Universal Robots URScript: script_ur5e.urscript

def ur5e_dibujar():
  textmsg("=== UR5e: inicio del programa ===")
  q_home = get_actual_joint_positions()
  textmsg("UR5e HOME guardado")
  # === Ir al origen calibrado: UR5e ===
  textmsg("UR5e - yendo al origen calibrado")
  x0 = 0.68387
  y0 = -0.03000
  z_mesa = 0.00221
  rx = 2.48100
  ry = -1.92700
  rz = 0.00000
  # Primero se acerca por arriba; nunca va directamente a la Z baja.
  movel(p[x0, y0, z_mesa+0.06000, rx, ry, rz], a=0.03, v=0.05)
  sleep(0.3)
  # === Detección única de superficie por fuerza: UR5e ===
  textmsg("UR5e - Detectando superficie una sola vez...")
  zero_ftsensor()
  sleep(0.5)
  i_f = 0
  while (force() < 2.000 and i_f < 2000):
    speedl([0, 0, -0.00800, 0, 0, 0], 0.25, 0.02)
    i_f = i_f + 1
  end
  stopl(3.0)
  sleep(0.2)
  if (i_f >= 2000):
    popup("UR5e: No se detectó superficie. Revisa posición inicial y F_UMBRAL.", error=True)
    halt
  end
  z_contacto = get_actual_tcp_pose()[2]
  z_dibujo = z_contacto + 0.00150
  textmsg("UR5e - z_contacto=", z_contacto)
  textmsg("UR5e - z_dibujo=", z_dibujo)
  movel(p[x0, y0, z_dibujo+0.02500, rx, ry, rz], a=0.03, v=0.04)
  sleep(0.2)
  # === Dibujo - UR5e - 3 trazos ===

  # --- Trazo 1 / 3 ---
  textmsg("UR5e - Trazo 1 de 3")
  movel(p[x0+0.01300, y0+-0.00696, z_dibujo+0.02500, rx, ry, rz], a=0.03, v=0.04)
  movel(p[x0+0.01300, y0+-0.00696, z_dibujo, rx, ry, rz], a=0.006, v=0.002)
  movel(p[x0+0.01269, y0+-0.00665, z_dibujo, rx, ry, rz], a=0.008, v=0.025, r=0.0002)
  movel(p[x0+0.01114, y0+-0.00665, z_dibujo, rx, ry, rz], a=0.008, v=0.025, r=0.0002)
  movel(p[x0+0.00990, y0+-0.00882, z_dibujo, rx, ry, rz], a=0.008, v=0.025, r=0.0002)
  movel(p[x0+0.00743, y0+-0.01130, z_dibujo, rx, ry, rz], a=0.008, v=0.025, r=0.0002)
  movel(p[x0+0.00464, y0+-0.01285, z_dibujo, rx, ry, rz], a=0.008, v=0.025, r=0.0002)
  movel(p[x0+0.00155, y0+-0.01346, z_dibujo, rx, ry, rz], a=0.008, v=0.025, r=0.0002)
  movel(p[x0+0.00124, y0+-0.01377, z_dibujo, rx, ry, rz], a=0.008, v=0.025, r=0.0002)
  movel(p[x0+0.00124, y0+-0.02182, z_dibujo, rx, ry, rz], a=0.008, v=0.025, r=0.0002)
  movel(p[x0+0.00217, y0+-0.02430, z_dibujo, rx, ry, rz], a=0.008, v=0.025, r=0.0002)
  movel(p[x0+0.00557, y0+-0.02801, z_dibujo, rx, ry, rz], a=0.008, v=0.025, r=0.0002)
  movel(p[x0+0.00960, y0+-0.02956, z_dibujo, rx, ry, rz], a=0.008, v=0.025, r=0.0002)
  movel(p[x0+0.01238, y0+-0.02956, z_dibujo, rx, ry, rz], a=0.008, v=0.025, r=0.0002)
  movel(p[x0+0.01269, y0+-0.02925, z_dibujo, rx, ry, rz], a=0.008, v=0.025, r=0.0002)
  movel(p[x0+0.01486, y0+-0.02894, z_dibujo, rx, ry, rz], a=0.008, v=0.025, r=0.0002)
  movel(p[x0+0.01888, y0+-0.02677, z_dibujo, rx, ry, rz], a=0.008, v=0.025, r=0.0002)
  movel(p[x0+0.02229, y0+-0.02306, z_dibujo, rx, ry, rz], a=0.008, v=0.025, r=0.0002)
  movel(p[x0+0.02383, y0+-0.01935, z_dibujo, rx, ry, rz], a=0.008, v=0.025, r=0.0002)
  movel(p[x0+0.02383, y0+-0.01532, z_dibujo, rx, ry, rz], a=0.008, v=0.025, r=0.0002)
  movel(p[x0+0.02229, y0+-0.01192, z_dibujo, rx, ry, rz], a=0.008, v=0.025, r=0.0002)
  movel(p[x0+0.01888, y0+-0.00882, z_dibujo, rx, ry, rz], a=0.008, v=0.025, r=0.0002)
  movel(p[x0+0.01331, y0+-0.00696, z_dibujo, rx, ry, rz], a=0.008, v=0.025, r=0.0002)
  movel(p[x0+0.01331, y0+-0.00696, z_dibujo+0.02500, rx, ry, rz], a=0.03, v=0.04)

  # --- Trazo 2 / 3 ---
  textmsg("UR5e - Trazo 2 de 3")
  movel(p[x0+0.02198, y0+0.01625, z_dibujo+0.02500, rx, ry, rz], a=0.03, v=0.04)
  movel(p[x0+0.02198, y0+0.01625, z_dibujo, rx, ry, rz], a=0.006, v=0.002)
  movel(p[x0+0.02167, y0+0.01656, z_dibujo, rx, ry, rz], a=0.008, v=0.025, r=0.0002)
  movel(p[x0+0.01733, y0+0.01656, z_dibujo, rx, ry, rz], a=0.008, v=0.025, r=0.0002)
  movel(p[x0+0.01455, y0+0.01532, z_dibujo, rx, ry, rz], a=0.008, v=0.025, r=0.0002)
  movel(p[x0+0.01269, y0+0.01377, z_dibujo, rx, ry, rz], a=0.008, v=0.025, r=0.0002)
  movel(p[x0+0.00836, y0+0.00789, z_dibujo, rx, ry, rz], a=0.008, v=0.025, r=0.0002)
  movel(p[x0+0.00836, y0+0.00727, z_dibujo, rx, ry, rz], a=0.008, v=0.025, r=0.0002)
  movel(p[x0+0.01052, y0+0.00480, z_dibujo, rx, ry, rz], a=0.008, v=0.025, r=0.0002)
  movel(p[x0+0.01176, y0+0.00201, z_dibujo, rx, ry, rz], a=0.008, v=0.025, r=0.0002)
  movel(p[x0+0.01176, y0+0.00077, z_dibujo, rx, ry, rz], a=0.008, v=0.025, r=0.0002)
  movel(p[x0+0.01207, y0+0.00046, z_dibujo, rx, ry, rz], a=0.008, v=0.025, r=0.0002)
  movel(p[x0+0.01207, y0+-0.00418, z_dibujo, rx, ry, rz], a=0.008, v=0.025, r=0.0002)
  movel(p[x0+0.01919, y0+-0.00665, z_dibujo, rx, ry, rz], a=0.008, v=0.025, r=0.0002)
  movel(p[x0+0.02260, y0+-0.00665, z_dibujo, rx, ry, rz], a=0.008, v=0.025, r=0.0002)
  movel(p[x0+0.02631, y0+-0.00511, z_dibujo, rx, ry, rz], a=0.008, v=0.025, r=0.0002)
  movel(p[x0+0.02940, y0+-0.00170, z_dibujo, rx, ry, rz], a=0.008, v=0.025, r=0.0002)
  movel(p[x0+0.03064, y0+0.00201, z_dibujo, rx, ry, rz], a=0.008, v=0.025, r=0.0002)
  movel(p[x0+0.03064, y0+0.00635, z_dibujo, rx, ry, rz], a=0.008, v=0.025, r=0.0002)
  movel(p[x0+0.03002, y0+0.00851, z_dibujo, rx, ry, rz], a=0.008, v=0.025, r=0.0002)
  movel(p[x0+0.02879, y0+0.01099, z_dibujo, rx, ry, rz], a=0.008, v=0.025, r=0.0002)
  movel(p[x0+0.02538, y0+0.01470, z_dibujo, rx, ry, rz], a=0.008, v=0.025, r=0.0002)
  movel(p[x0+0.02352, y0+0.01594, z_dibujo, rx, ry, rz], a=0.008, v=0.025, r=0.0002)
  movel(p[x0+0.02229, y0+0.01625, z_dibujo, rx, ry, rz], a=0.008, v=0.025, r=0.0002)
  movel(p[x0+0.02229, y0+0.01625, z_dibujo+0.02500, rx, ry, rz], a=0.03, v=0.04)

  # --- Trazo 3 / 3 ---
  textmsg("UR5e - Trazo 3 de 3")
  movel(p[x0+-0.01857, y0+0.01656, z_dibujo+0.02500, rx, ry, rz], a=0.03, v=0.04)
  movel(p[x0+-0.01857, y0+0.01656, z_dibujo, rx, ry, rz], a=0.006, v=0.002)
  movel(p[x0+-0.01888, y0+0.01687, z_dibujo, rx, ry, rz], a=0.008, v=0.025, r=0.0002)
  movel(p[x0+-0.02136, y0+0.01656, z_dibujo, rx, ry, rz], a=0.008, v=0.025, r=0.0002)
  movel(p[x0+-0.02476, y0+0.01501, z_dibujo, rx, ry, rz], a=0.008, v=0.025, r=0.0002)
  movel(p[x0+-0.02848, y0+0.01099, z_dibujo, rx, ry, rz], a=0.008, v=0.025, r=0.0002)
  movel(p[x0+-0.02971, y0+0.00851, z_dibujo, rx, ry, rz], a=0.008, v=0.025, r=0.0002)
  movel(p[x0+-0.03033, y0+0.00635, z_dibujo, rx, ry, rz], a=0.008, v=0.025, r=0.0002)
  movel(p[x0+-0.03033, y0+0.00170, z_dibujo, rx, ry, rz], a=0.008, v=0.025, r=0.0002)
  movel(p[x0+-0.02879, y0+-0.00232, z_dibujo, rx, ry, rz], a=0.008, v=0.025, r=0.0002)
  movel(p[x0+-0.02600, y0+-0.00511, z_dibujo, rx, ry, rz], a=0.008, v=0.025, r=0.0002)
  movel(p[x0+-0.02260, y0+-0.00665, z_dibujo, rx, ry, rz], a=0.008, v=0.025, r=0.0002)
  movel(p[x0+-0.01888, y0+-0.00665, z_dibujo, rx, ry, rz], a=0.008, v=0.025, r=0.0002)
  movel(p[x0+-0.01207, y0+-0.00449, z_dibujo, rx, ry, rz], a=0.008, v=0.025, r=0.0002)
  movel(p[x0+-0.01176, y0+-0.00418, z_dibujo, rx, ry, rz], a=0.008, v=0.025, r=0.0002)
  movel(p[x0+-0.01176, y0+0.00077, z_dibujo, rx, ry, rz], a=0.008, v=0.025, r=0.0002)
  movel(p[x0+-0.01114, y0+0.00294, z_dibujo, rx, ry, rz], a=0.008, v=0.025, r=0.0002)
  movel(p[x0+-0.00990, y0+0.00542, z_dibujo, rx, ry, rz], a=0.008, v=0.025, r=0.0002)
  movel(p[x0+-0.00805, y0+0.00727, z_dibujo, rx, ry, rz], a=0.008, v=0.025, r=0.0002)
  movel(p[x0+-0.00805, y0+0.00789, z_dibujo, rx, ry, rz], a=0.008, v=0.025, r=0.0002)
  movel(p[x0+-0.01114, y0+0.01223, z_dibujo, rx, ry, rz], a=0.008, v=0.025, r=0.0002)
  movel(p[x0+-0.01424, y0+0.01532, z_dibujo, rx, ry, rz], a=0.008, v=0.025, r=0.0002)
  movel(p[x0+-0.01702, y0+0.01656, z_dibujo, rx, ry, rz], a=0.008, v=0.025, r=0.0002)
  movel(p[x0+-0.01826, y0+0.01656, z_dibujo, rx, ry, rz], a=0.008, v=0.025, r=0.0002)
  movel(p[x0+-0.01826, y0+0.01656, z_dibujo+0.02500, rx, ry, rz], a=0.03, v=0.04)

  textmsg("UR5e - Dibujo completado")
  textmsg("UR5e - Volviendo a HOME")
  movej(q_home, a=0.03, v=0.05)
  textmsg("UR5e - En HOME. Programa completado")
end
ur5e_dibujar()
